Universal Robots PolyScope program: projeto_final_13062.urp

Program projeto_final_13062 (createdIn=3.4.5.437 lastSavedIn=3.4.5.437 directory=/programs/usbdisk installation=default robotSerialNumber=2017357015)
Calibrated DH parameters: a=[0.000021, -0.261063, -0.376363, 0.000077, 0.000104, 0]; d=[0.089312, 121.214456, -102.904559, -18.199769, 0.094928, 0.082537]; alpha=[1.569843, -0.002771, -0.006062, 1.56958, -1.570059, 0]; deltaTheta=[0.000006, -0.909999, 0.623282, 0.286705, -0.000096, 0.00002]
InitVariablesNode
BeforeStart
  Folder cria_variaveis_pos
    phome := Base
    phand := Base
    pplay := Base
    Script: teach_mode()
    ppickx := 0
    ppicky := 0
    pplacex := 0
    pplacey := 0
    ppickxmod := 0
    ppickymod := 0
    actual_pose := [0,0,0,0,0,0]
    picktheta := 0
    placetheta := 0
    pplacexmod := 0
    pplaceymod := 0
    tcp_pose := Base
    z0_place := -0.228
    waiting := 0
    zpick := 0.0095
    z0_pick := -0.078
    robot_turn := False
    bigdouble := False
    pass := False
    sinal_enviado := False
    game_over := False
    PCam_board := Cam_Pose_Board
    PCam_Hand := Cam_Pose_Hand
    Script: write_port_bit(21, False )
  Folder define_pos_padroes
    Popup Message (haltProgram=false message=Mova o robo para a posicao home e clique em continuar.)
    Wait Sleep waitTime=0.5
    Folder Folder
      Script: end_teach_mode()
      actual_pose := get_actual_joint_positions()
      Script: actual_pose[5]=0
      Script: movej(actual_pose)
    Script: teach_mode()
    Script: phome=get_actual_tcp_pose()
    Popup Message (haltProgram=false message=mova o robo para a posicao hand e clique em continuar.)
    Script: phand=get_actual_tcp_pose()
    Popup Message (haltProgram=false message=Mova o robo para a posicao play e clique em continuar)
    Script: pplay=get_actual_tcp_pose()
  Script: end_teach_mode()
  Script: movej(phome)
Robot Program (runOnlyOnce=false motionType=MoveJ speed=1.047198 acceleration=1.396263 useActiveTCP=false)
  Folder wait_init [hidden by the author, left out]
  If pass≟ False
    waiting := 1
    pass_test := False
    Folder Main
      If waiting_player≟ True
        If robot_turn≟ True
          Call pick_hand
        Else 
          Wait Sleep waitTime=0.01
      ElseIf piece_picked≟ True
        Call place_piece
      ElseIf piece_placed≟ True
        Call wait_player
        robot_turn := False
  Else 
    Wait Sleep waitTime=0.01
    pass_test := True
    Call wait_player
    piece_placed := True
SubProgram -> wait_player
SubProgram -> pick_hand
SubProgram -> place_piece
Thread Thread_1 (runOnlyOnce=false trackProgramExecution=false)
  Folder Folder
    Script file /programs/converte_num.script
      | def converte_num(num):
      |  if num >=32767:
      |   num=num-65536
      |  end
      |  return num
      | end
    Script file /programs/pick_values_modbus_check.script_bak
      | pass=read_port_bit(18)
      | game_over=read_port_bit(19)
      | 
      | #registradores
      | ppickx = converte_num(read_port_register(128))/1000
      | ppicky=converte_num(read_port_register(129))/1000
      | pplacex=converte_num(read_port_register(130))/1000
      | pplacey=converte_num(read_port_register(131))/1000
      | picktheta=converte_num(read_port_register(132))/1000
      | placetheta=converte_num(read_port_register(133))/1000
      | 
      | #booleanos
      | bigdouble=read_port_bit(17)
      | sinal_enviado=read_port_bit(20)
    Script file /programs/calcula_tcp.script_bak
      | ppickxmod=ppickx-0.02*cos(picktheta)
      | ppickymod=ppicky+0.02*sin(picktheta)
      | pplacexmod=pplacex-0.02*cos(placetheta)
      | pplaceymod=pplacey+0.02*sin(placetheta)
    If digital_in[1]≟ True  and piece_placed≟ True
      piece_placed := False
      Script: write_port_bit(21, True )
      Wait Condition expression=read_port_bit(20)
      Script: write_port_bit(21, False )
      Wait Sleep waitTime=2
      Script file /programs/pick_values_modbus_check.script_bak
        | (same text as the earlier copy of this file)
      Script file /programs/calcula_tcp.script_bak
        | ppickxmod=ppickx-0.02*cos(picktheta)
        | ppickymod=ppicky+0.02*sin(picktheta)
        | pplacexmod=pplacex-0.02*cos(placetheta)
        | pplaceymod=pplacey+0.02*sin(placetheta)
      game_over_var_1 := False
      Wait Sleep waitTime=0.01
      robot_turn := True
    Wait Sleep waitTime=0.01
    If game_over≟ True  and game_over_var_1≟ True
      Popup Message (haltProgram=true message=FIM DE JOGO!!)
SubProgram pick_hand (keepSynchronizedWithDisk=false trackProgramExecution=false)
  waiting_player := False
  Script: movel(phand)
  Set DigitalOutput pin=tool_out[0]; digitalValue=0
  Set DigitalOutput pin=tool_out[1]; digitalValue=1
  Wait Sleep waitTime=0.2
  Script: movej(pose_add(p[ppickx,ppicky,z0_pick,0,0,0],Cam_Pose_Hand))
  leitura_test := pose_add(p[ppickx,ppicky,z0_pick,0,0,0],Cam_Pose_Hand)
  Wait Sleep waitTime=0.1
  If bigdouble≟ False
    actual_pose := get_actual_joint_positions()
    Script: actual_pose[5]=actual_pose[5]+picktheta
    Script: movej(actual_pose)
    tcp_pose := get_actual_tcp_pose()
    Script: tcp_pose[2]=tcp_pose[2]-zpick
    Script: movej(tcp_pose)
    Set DigitalOutput pin=tool_out[1]; digitalValue=0
    Set DigitalOutput pin=tool_out[0]; digitalValue=1
    Wait Sleep waitTime=0.5
    tcp_pose := get_actual_tcp_pose()
    Script: tcp_pose[2]=tcp_pose[2]+zpick
    Script: movej(tcp_pose)
    Folder Folder
      actual_pose := get_actual_joint_positions()
      Script: actual_pose[5]=0
      Script: movej(actual_pose)
    Script: movel(phand)
    piece_picked := True   [initializeExpression=False]
  Else 
    Script: movej(pose_add(p[ppickxmod,ppickymod,z0_pick,0,0,0],Cam_Pose_Hand))
    actual_pose := get_actual_joint_positions()
    Script: actual_pose[5]=actual_pose[5]+picktheta+1.57
    Script: movej(actual_pose)
    tcp_pose := get_actual_tcp_pose()
    Script: tcp_pose[2]=tcp_pose[2]-zpick
    Script: movej(tcp_pose)
    Wait Sleep waitTime=0.1
    Set DigitalOutput pin=tool_out[1]; digitalValue=0
    Set DigitalOutput pin=tool_out[0]; digitalValue=1
    Wait Sleep waitTime=0.3
    Folder Folder
      tcp_pose := get_actual_tcp_pose()
      Script: tcp_pose[2]=tcp_pose[2]+zpick
      Script: movej(tcp_pose)
      actual_pose := get_actual_joint_positions()
      Script: actual_pose[5]=0
      Script: movej(actual_pose)
    Script: movej(phand)
    piece_picked := True
SubProgram place_piece (keepSynchronizedWithDisk=false trackProgramExecution=false)
  piece_picked := False
  Script: movej(pplay)
  Wait Sleep waitTime=0.1
  Folder Folder
    actual_pose := get_actual_joint_positions()
    Script: actual_pose[5]=0
    Script: movej(actual_pose)
  Script: movej(pose_add(p[pplacex,pplacey,z0_place,0,0,0],Cam_Pose_Board))
  leitura_test := pose_add(p[pplacex,pplacey,z0_place,0,0,0],Cam_Pose_Board)
  Wait Sleep waitTime=0.1
  If bigdouble≟ False
    actual_pose := get_actual_joint_positions()
    Script: actual_pose[5]=actual_pose[5]+placetheta
    Wait Sleep waitTime=0.1
    Script: movej(actual_pose)
    tcp_pose := get_actual_tcp_pose()
    Script: tcp_pose[2]=tcp_pose[2]-zpick
    Script: movej(tcp_pose)
    Set DigitalOutput pin=tool_out[0]; digitalValue=0
    Set DigitalOutput pin=tool_out[1]; digitalValue=1
    Wait Sleep waitTime=0.2
    tcp_pose := get_actual_tcp_pose()
    Script: tcp_pose[2]=tcp_pose[2]+3*zpick
    Script: movej(tcp_pose)
    Folder Folder
      actual_pose := get_actual_joint_positions()
      Script: actual_pose[5]=0
      Script: movej(actual_pose)
  Else 
    Script: movej(pose_add(p[pplacexmod,pplaceymod,z0_place,0,0,0],Cam_Pose_Board))
    actual_pose := get_actual_joint_positions()
    Script: actual_pose[5]=actual_pose[5]+placetheta+1.57
    Script: movej(actual_pose)
    tcp_pose := get_actual_tcp_pose()
    Script: tcp_pose[2]=tcp_pose[2]-zpick
    Script: movej(tcp_pose)
    Wait Sleep waitTime=0.1
    Set DigitalOutput pin=tool_out[0]; digitalValue=0
    Set DigitalOutput pin=tool_out[1]; digitalValue=1
    Wait Sleep waitTime=0.3
    tcp_pose := get_actual_tcp_pose()
    Script: tcp_pose[2]=tcp_pose[2]+3*zpick
    Script: movej(tcp_pose)
    Folder Folder
      actual_pose := get_actual_joint_positions()
      Script: actual_pose[5]=0
      Script: movej(actual_pose)
  Wait Sleep waitTime=0.2
  Folder Folder
    actual_pose := get_actual_joint_positions()
    Script: actual_pose[5]=0
    Script: movej(actual_pose)
  Script: movel(pplay)
  Set DigitalOutput pin=tool_out[1]; digitalValue=0
  Set DigitalOutput pin=tool_out[0]; digitalValue=1
  game_over_var_1 := True   [initializeExpression=False]
  piece_placed := True   [initializeExpression=True]
  Wait Sleep waitTime=0.2
SubProgram wait_player (keepSynchronizedWithDisk=false trackProgramExecution=false)
  If waiting≟1 and pass_test≟ True
    Force Simple feature=Base; selection=[0, 0, 1, 0, 0, 0]; wrench=[0, 0, -30, 0, 0, 0]; limitsForce=[0.15, 0.15, 0.15, 1.047198, 1.047198, 1.047198]; limitsMotion=[0.1, 0.1, 0.1, 0.349066, 0.349066, 0.349066]
      Wait Sleep waitTime=2
    tcp_pose := get_actual_tcp_pose()
    Script: tcp_pose[2]=tcp_pose[2]+0.05
    Script: movej(tcp_pose)
    Force Simple feature=Base; selection=[0, 0, 1, 0, 0, 0]; wrench=[0, 0, -30, 0, 0, 0]; limitsForce=[0.15, 0.15, 0.15, 1.047198, 1.047198, 1.047198]; limitsMotion=[0.1, 0.1, 0.1, 0.349066, 0.349066, 0.349066]
      Wait Sleep waitTime=2
    Script: movej(phome)
    Wait Sleep waitTime=0.01
    waiting_player := True
    waiting := 0
  Else 
    Script: movej(phome)
    Wait Sleep waitTime=0.01
    waiting_player := True
